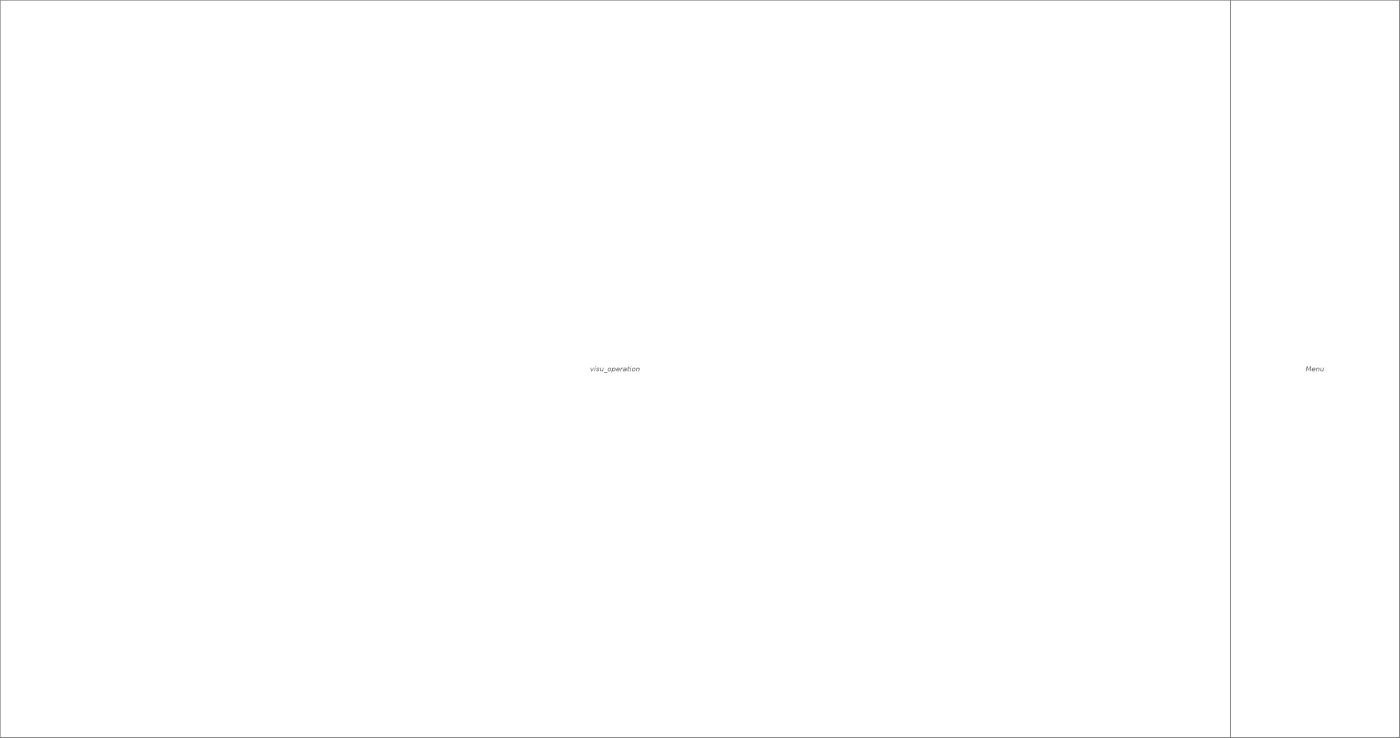
VISUALIZATION visu_main  // 2048x1080
    Frame (0,0 1800x1080), frame switch variable: G_HMI.iMainFrame
        shows visu_operation()
        shows visu_buffer()
        shows visu_loading()
        shows visu_working()
        shows v_alarm()
        shows v_IO_fixtureClamp()
    Frame (1800,0 248x1080), frame switch variable: G_HMI.iMainFrame
        shows Menu()
        shows visu_working()
        shows v_IO_fixtureClamp()
        shows visu_buffer()
        shows visu_loading()
        shows v_alarm()
END_VISUALIZATION

(* stored: Version 1.1.0.1, ProductVersion 3.1.4024.12
   Visu visu_main: Id {27f18664-69ba-41bf-9a81-29f5cd36101a} *)
